// TwinCAT 3 PLC project MAIN
// ProgramVersion: 3.1.4023.0
// libraries:
//   Tc2_ModbusRTU, * (Beckhoff Automation GmbH)
//   Tc2_ModbusSrv, * (Beckhoff Automation GmbH)
//   Tc2_Standard, * (Beckhoff Automation GmbH)
//   Tc2_System, * (Beckhoff Automation GmbH)
//   Tc3_Module, * (Beckhoff Automation GmbH)
// project tree:
//   DUTs/ FUSSION.TcDUT, Inverter_SUN2000.TcDUT
//   / PlcTask.TcTTO
//   POUs/ FB_ModbusMaster_FUSSION.TcPOU, FB_ModbusMaster_Inverter.TcPOU, MAIN.TcPOU

CONFIGURATION MAIN
    RESOURCE PLC ON TwinCAT3
        TASK PlcTask(INTERVAL := T#10ms, PRIORITY := 20);
        PROGRAM MAIN WITH PlcTask : MAIN;
    END_RESOURCE
END_CONFIGURATION

// ---- DUTs/FUSSION.TcDUT
TYPE FUSSION :
STRUCT
	IPAddr		: STRING:= '127.0.0.1';
	IDSlave		: BYTE:= 255;
	TCPPort		: UINT:= 500;
	
	//--------------- LECTURA INPUT REGISTERS ---------------
	uiAddress_InputRegisters 		: ARRAY [1..19] OF UINT:= [1, 2, 3, 4, 5, 256, 257, 258, 259, 260, 261, 36864, 36865, 36866, 36867, 36868, 36869, 36870, 36871];
	uiRaw_InputRegisters 			: ARRAY [1..19] OF UINT;
	
	FSM_State_Outlet1	: UINT;
	Power_Outlet1		: UDINT;
	Energy_Outlet1		: UDINT;
	FSM_State_Outlet2	: UDINT;
	Power_Outlet2		: UDINT;
	Energy_Outlet2		: UDINT;
	Power_Phase1_Total	: UDINT;
	Power_Phase2_Total	: UDINT;
	Power_Phase3_Total	: UDINT;
	Number_Available_CPs: UDINT;
	
	//--------------- LECTURA HOLDING REGISTERS ---------------
	uiAddress_HoldingRegisters 		: ARRAY [1..18] OF WORD:= [32768,32769, 32770, 32771, 32772, 32773, 32774, 32775, 32776, 32777, 32784, 32785, 36864, 36865, 36866, 36867, 36868, 36869];
	
	uiRaw_HoldingRegisters			: ARRAY [1..18] OF UINT; // Variables leidas de Modbus para escritura en pyads
	Power_Phase1_Max_Outlet1		: UDINT;
	Power_Phase2_Max_Outlet1		: UDINT;
	Power_Phase3_Max_Outlet1		: UDINT;
	Power_Phase1_Max_Outlet2		: UDINT;
	Power_Phase2_Max_Outlet2		: UDINT;
	Power_Phase3_Max_Outlet2		: UDINT;
	Power_Phase1_Total_Max			: UDINT;
	Power_Phase2_Total_Max			: UDINT;
	Power_Phase3_Total_Max			: UDINT;
	
	uiRaw_HoldingRegisters_write	: ARRAY [1..18] OF UINT; // Variables recibidas para escritura en Modbus
		
	//Power_Phase1_Max_Outlet1_write	: UDINT;
	//Power_Phase2_Max_Outlet1_write	: UDINT;
	//Power_Phase3_Max_Outlet1_write	: UDINT;
	//Power_Phase1_Max_Outlet2_write	: UDINT;
	//Power_Phase2_Max_Outlet2_write	: UDINT;
	//Power_Phase3_Max_Outlet2_write	: UDINT;
	//Power_Phase1_Total_Max_write	: UDINT;
	//Power_Phase2_Total_Max_write	: UDINT;
	//Power_Phase3_Total_Max_write	: UDINT;
	
		
END_STRUCT
END_TYPE

// ---- DUTs/Inverter_SUN2000.TcDUT
TYPE Inverter_SUN2000 :
STRUCT
	IDSlave		: BYTE:= 255;
	TCPPort		: UINT:= 500;
	
	//--------------- LECTURA ALARMAS ---------------
	uiAddress_Alarm 		: ARRAY [1..11] OF UINT:= [50000, 50001, 50002, 50003, 50004, 50005, 50006, 50007, 50008, 50009, 50016];
	uiRaw_Alarm 			: ARRAY [1..11] OF UINT;
	
	// 50000
	Software_Ver_Unmatch_1	:	BOOL;
	Upgrade_Failed_1		:	BOOL;
	Flash_Fault_1			:	BOOL;
	// 50001
	Software_Ver_Unmatch_2	:	BOOL;
	Software_Ver_Unmatch_3	:	BOOL;
	System_Fault_1			:	BOOL;
	System_Fault_27			:	BOOL;
	Abnormal_Inv_Circuit_20	:	BOOL;
	Abnormal_Resid_Cur_1	:	BOOL;
	Cabinet_Overtemp_1		:	BOOL;
	System_Fault_28			:	BOOL;
	Fan_Fault_1				:	BOOL;
	Abnormal_SPI_Comm_1		:	BOOL;
	System_Fault_29			:	BOOL;
	//50002
	Low_Insulation_Res_1	:	BOOL;
	AFCI_Self_test_Fault_1	:	BOOL;
	DC_Arc_Fault_1			:	BOOL;
	AFCI_Self_test_Fault_2	:	BOOL;
	AFCI_Self_test_Fault_3	:	BOOL;
	System_Fault_30			:	BOOL;
	System_Fault_31			:	BOOL;
	String_3_Reversed_1		:	BOOL;
	DC_Arc_Fault_2			:	BOOL;
	DC_Arc_Fault_3			:	BOOL;
	DC_Arc_Fault_4			:	BOOL;
	System_Fault_23			:	BOOL;
	// 50003
	String_1_Reversed_1		:	BOOL;
	String_2_Reversed_1		:	BOOL;
	Abnormal_DC_Circuit_12	:	BOOL;
	String_4_Reversed_1		:	BOOL;
	String_5_Reversed_1		:	BOOL;
	String_6_Reversed_1		:	BOOL;
	High_DC_Input_Volt_1	:	BOOL;
	High_DC_Input_Volt_2	:	BOOL;
	High_DC_Input_Volt_3	:	BOOL;
	High_DC_Input_Volt_4	:	BOOL;
	Abnormal_DC_Circuit_15	:	BOOL;
	// 50004
	String_1_Reversed_2		:	BOOL;
	String_2_Reversed_2		:	BOOL;
	String_7_Reversed_1		:	BOOL;
	String_7_Reversed_2		:	BOOL;
	String_8_Reversed_1		:	BOOL;
	String_8_Reversed_2		:	BOOL;
	String_3_Reversed_2		:	BOOL;
	String_4_Reversed_2		:	BOOL;
	String_5_Reversed_2		:	BOOL;
	String_6_Reversed_2		:	BOOL;
	// 50005
	Abnormal_DC_Circuit_3	:	BOOL;
	Abnormal_Auxiliary_power_4	:	BOOL;
	Abnormal_DC_Circuit_10	:	BOOL;
	Abnormal_DC_Circuit_11	:	BOOL;
	Abnormal_DC_Circuit_30	:	BOOL;
	// 50006
	System_Fault_3			:	BOOL;
	Abnormal_Inv_Circuit_13	:	BOOL;
	Abnormal_Inv_Circuit_14	:	BOOL;
	// 50007
	Abnormal_Inv_Circuit_16	:	BOOL;
	System_Fault_21			:	BOOL;
	// 50008
	Abnormal_Grid_Volt_4	:	BOOL;
	Abnormal_Grid_Volt_16	:	BOOL;
	Frequency_Abnormal_2	:	BOOL;
	Frequency_Abnormal_4	:	BOOL;
	Abnormal_Grid_Volt_28	:	BOOL;
	Abnormal_Grid_Volt_29	:	BOOL;
	Abnormal_Ground_1		:	BOOL;
	Abnormal_Grid_Volt_26	:	BOOL;
	Frequency_Abnormal_5	:	BOOL;
	// 50009
	Abnormal_Grid_Volt_31	:	BOOL;
	Abnormal_Grid_Volt_32	:	BOOL;
	Abnormal_Grid_Volt_33	:	BOOL;
	Abnormal_Grid_Volt_19	:	BOOL;
	// 50016
	Abnormal_String_1_1		:	BOOL;
	Abnormal_String_2_1		:	BOOL;
	Abnormal_String_3_1		:	BOOL;
	Abnormal_String_4_1		:	BOOL;
	Abnormal_String_5_1		:	BOOL;
	Abnormal_String_6_1		:	BOOL;
	Abnormal_String_7_1		:	BOOL;
	Abnormal_String_8_1		:	BOOL;
	
	//--------------- LECTURA MEDIDAS ---------------
	//Falta por determinar que variables queremos medir.
	uiAddress_Signal 		: ARRAY [1..137] OF UINT:= [32001,32002,32003,32200,32262,32263,32264,32265,32266,32267,32268,32269,32270,32271,32272,32273,32274,32275,32276,32277,
														32278,32279,32280,32281,32282,32283,32284,32285,32286,32287,32288,32290,32292,32294,32296,32298,32300,32302,32304,32306,
														32314,32315,32316,32317,32320,32321,32321,32321,32322,32323,32325,32327,32343,32345,32347,32349,32351,32353,32355,32357,
														33022,33024,33026,33070,40000,40117,40118,40119,40120,40121,40122,40123,40124,40125,40133,40154,40200,40201,40232,40234,
														40235,40236,40237,42045,42047,42049,42051,42053,42055,42057,42059,42061,42063,42064,42065,42066,42067,42068,42069,42070,
														42071,42072,42074,42075,42083,42084,42085,42086,42087,42089,42090,42091,42092,42093,42094,42095,42096,42097,42101,42151,
														42152,42154,42155,42157,42158,42160,42161,42174,42300,42301,42302,42303,42304,42305,42320,42321,42333];
	uiRaw_Signal			: ARRAY [1..137] OF UINT;
END_STRUCT
END_TYPE

// ---- POUs/MAIN.TcPOU
PROGRAM MAIN
VAR
	FUSSION: FB_ModbusMaster_FUSSION;
	Inverter: FB_ModbusMaster_Inverter;
	Enable: BOOL:= TRUE;
	
	salida_pyads_InputRegisters: ARRAY[1..10] OF UINT;
	salida_pyads_HoldingsRegisters: ARRAY[1..9] OF UINT;
	entrada_pyads: ARRAY[1..9] OF UINT;
	flag_entrada_pyads: BOOL;
END_VAR

FUSSION(
	bEnable:= Enable, 
	entrada_pyads:= entrada_pyads, 
	flag_entrada_pyads:= flag_entrada_pyads, 
	salida_pyads_InputRegisters=> salida_pyads_InputRegisters, 
	salida_pyads_HoldingsRegisters=> salida_pyads_HoldingsRegisters);
	
//Inverter(bEnable:= Enable);

END_PROGRAM

// ---- POUs/FB_ModbusMaster_FUSSION.TcPOU
FUNCTION_BLOCK FB_ModbusMaster_FUSSION
VAR_INPUT
	bEnable			: BOOL;
	entrada_pyads: ARRAY[1..9] OF UINT; // Variables recibidas para escritura en Modbus
END_VAR
VAR
	iPaso			: INT;
	fbReadRegs		: FB_MBReadRegs;
	fbReadInputRegs : FB_MBReadInputRegs;
	bOcupado		: BOOL;
	
	Data_FUSSION : FUSSION;
	bAddrCount		: BYTE:= 1;
	bAddrCount2: BYTE;
	bOcupado2: BOOL;
	counter: BYTE := 1;
	fbWriteRegs: FB_MBWriteRegs;
	bOcupado3: BOOL;
	
END_VAR
VAR_OUTPUT
	salida_pyads_InputRegisters: ARRAY[1..10] OF UINT;
	salida_pyads_HoldingsRegisters: ARRAY[1..9] OF UINT;
END_VAR
VAR_IN_OUT
	flag_entrada_pyads: BOOL;
END_VAR

CASE iPaso OF
0:	//Inicio
	fbReadRegs(bExecute := FALSE);
	fbReadInputRegs(bExecute := FALSE);
	IF bEnable THEN
		iPaso := 1;
	END_IF

1: //Lectura Input Registers
	fbReadInputRegs(
			sIPAddr		:= Data_FUSSION.IPAddr, 
			nTCPPort	:= Data_FUSSION.TCPPort, 
			nUnitID		:= Data_FUSSION.IDSlave, 
			nQuantity	:= 1, 
			nMBAddr		:= Data_FUSSION.uiAddress_InputRegisters[bAddrCount],
			cbLength	:= SIZEOF(Data_FUSSION.uiRaw_InputRegisters[bAddrCount]),
			pDestAddr	:= ADR(Data_FUSSION.uiRaw_InputRegisters[bAddrCount]), 
			bExecute	:= TRUE, 
			tTimeout	:= T#1S, 
			bBusy		=> bOcupado, 
			bError		=> , 
			nErrId		=> , 
			cbRead		=> );
	IF NOT bOcupado THEN
		fbReadInputRegs(bExecute := FALSE);
		bAddrCount := bAddrCount+1;
		IF bAddrCount > 19 THEN
			bAddrCount := 1;
			bAddrCount2 := 1;
			iPaso := 4;	
		END_IF
	END_IF
	
3: //Lectura Holding Registers
	fbReadRegs(
		sIPAddr		:= Data_FUSSION.IPAddr, 
		nTCPPort	:= Data_FUSSION.TCPPort, 
		nUnitID		:= Data_FUSSION.IDSlave, 
		nQuantity	:= 1,
		nMBAddr		:= Data_FUSSION.uiAddress_HoldingRegisters[bAddrCount2],
		cbLength	:= SIZEOF(Data_FUSSION.uiRaw_HoldingRegisters[bAddrCount2]), 
		pDestAddr	:= ADR(Data_FUSSION.uiRaw_HoldingRegisters[bAddrCount2]), 
		bExecute	:= TRUE, 
		tTimeout	:= T#1S, 
		bBusy		=> bOcupado2, 
		bError		=> , 
		nErrId		=> , 
		cbRead		=> );
	IF NOT bOcupado2 THEN
		fbReadRegs(bExecute := FALSE);
		bAddrCount2 := bAddrCount2+1;
			IF bAddrCount2 > 18 THEN
				bAddrCount2 := 1;
				iPaso := 4;	
			END_IF
	END_IF

4: //Escalado Input Registers
	Data_FUSSION.FSM_State_Outlet1 		:= Data_FUSSION.uiRaw_InputRegisters[1]; // Little
	Data_FUSSION.Power_Outlet1			:= SHL(Data_FUSSION.uiRaw_InputRegisters[3], 8) + Data_FUSSION.uiRaw_InputRegisters[2];
	Data_FUSSION.Energy_Outlet1			:= SHL(Data_FUSSION.uiRaw_InputRegisters[5], 8) + Data_FUSSION.uiRaw_InputRegisters[4];
	Data_FUSSION.FSM_State_Outlet2		:= SHL(Data_FUSSION.uiRaw_InputRegisters[7], 8) + Data_FUSSION.uiRaw_InputRegisters[6];
	Data_FUSSION.Power_Outlet2			:= SHL(Data_FUSSION.uiRaw_InputRegisters[9], 8) + Data_FUSSION.uiRaw_InputRegisters[8];
	Data_FUSSION.Energy_Outlet2			:= SHL(Data_FUSSION.uiRaw_InputRegisters[11], 8) + Data_FUSSION.uiRaw_InputRegisters[10];
	Data_FUSSION.Power_Phase1_Total		:= SHL(Data_FUSSION.uiRaw_InputRegisters[12], 8) + Data_FUSSION.uiRaw_InputRegisters[13]; // Big
	Data_FUSSION.Power_Phase2_Total		:= SHL(Data_FUSSION.uiRaw_InputRegisters[14], 8) + Data_FUSSION.uiRaw_InputRegisters[15];
	Data_FUSSION.Power_Phase3_Total		:= SHL(Data_FUSSION.uiRaw_InputRegisters[16], 8) + Data_FUSSION.uiRaw_InputRegisters[17];
	Data_FUSSION.Number_Available_CPs 	:= SHL(Data_FUSSION.uiRaw_InputRegisters[18], 8) + Data_FUSSION.uiRaw_InputRegisters[19];
	
	//Temporales pyads
	salida_pyads_InputRegisters[1] 		:= Data_FUSSION.uiRaw_InputRegisters[1]; // Little
	salida_pyads_InputRegisters[2]		:= SHL(Data_FUSSION.uiRaw_InputRegisters[3], 8) + Data_FUSSION.uiRaw_InputRegisters[2];
	salida_pyads_InputRegisters[3]		:= SHL(Data_FUSSION.uiRaw_InputRegisters[5], 8) + Data_FUSSION.uiRaw_InputRegisters[4];
	salida_pyads_InputRegisters[4]		:= SHL(Data_FUSSION.uiRaw_InputRegisters[7], 8) + Data_FUSSION.uiRaw_InputRegisters[6];
	salida_pyads_InputRegisters[5]		:= SHL(Data_FUSSION.uiRaw_InputRegisters[9], 8) + Data_FUSSION.uiRaw_InputRegisters[8];
	salida_pyads_InputRegisters[6]		:= SHL(Data_FUSSION.uiRaw_InputRegisters[11], 8) + Data_FUSSION.uiRaw_InputRegisters[10];
	salida_pyads_InputRegisters[7]		:= SHL(Data_FUSSION.uiRaw_InputRegisters[12], 8) + Data_FUSSION.uiRaw_InputRegisters[13]; // Big
	salida_pyads_InputRegisters[8]		:= SHL(Data_FUSSION.uiRaw_InputRegisters[14], 8) + Data_FUSSION.uiRaw_InputRegisters[15];
	salida_pyads_InputRegisters[9]		:= SHL(Data_FUSSION.uiRaw_InputRegisters[16], 8) + Data_FUSSION.uiRaw_InputRegisters[17];
	salida_pyads_InputRegisters[10]	 	:= SHL(Data_FUSSION.uiRaw_InputRegisters[18], 8) + Data_FUSSION.uiRaw_InputRegisters[19];

	iPaso := 6;
	
5: //Escalado Holding Registers
	Data_FUSSION.Power_Phase1_Max_Outlet1	:= SHL(Data_FUSSION.uiRaw_HoldingRegisters[2], 8) + Data_FUSSION.uiRaw_HoldingRegisters[1]; // Little
	Data_FUSSION.Power_Phase2_Max_Outlet1	:= SHL(Data_FUSSION.uiRaw_HoldingRegisters[4], 8) + Data_FUSSION.uiRaw_HoldingRegisters[3];
	Data_FUSSION.Power_Phase3_Max_Outlet1	:= SHL(Data_FUSSION.uiRaw_HoldingRegisters[6], 8) + Data_FUSSION.uiRaw_HoldingRegisters[5];
	Data_FUSSION.Power_Phase1_Max_Outlet2	:= SHL(Data_FUSSION.uiRaw_HoldingRegisters[8], 8) + Data_FUSSION.uiRaw_HoldingRegisters[7];
	Data_FUSSION.Power_Phase2_Max_Outlet2	:= SHL(Data_FUSSION.uiRaw_HoldingRegisters[10], 8) + Data_FUSSION.uiRaw_HoldingRegisters[9];
	Data_FUSSION.Power_Phase3_Max_Outlet2	:= SHL(Data_FUSSION.uiRaw_HoldingRegisters[12], 8) + Data_FUSSION.uiRaw_HoldingRegisters[11];
	Data_FUSSION.Power_Phase1_Total_Max		:= SHL(Data_FUSSION.uiRaw_HoldingRegisters[13], 8) + Data_FUSSION.uiRaw_HoldingRegisters[14]; // Big
	Data_FUSSION.Power_Phase2_Total_Max		:= SHL(Data_FUSSION.uiRaw_HoldingRegisters[15], 8) + Data_FUSSION.uiRaw_HoldingRegisters[16];
	Data_FUSSION.Power_Phase3_Total_Max		:= SHL(Data_FUSSION.uiRaw_HoldingRegisters[17], 8) + Data_FUSSION.uiRaw_HoldingRegisters[18];
	
	//Temporales pyads
	salida_pyads_HoldingsRegisters[1]		:= SHL(Data_FUSSION.uiRaw_HoldingRegisters[2], 8) + Data_FUSSION.uiRaw_HoldingRegisters[1]; // Little
	salida_pyads_HoldingsRegisters[2]		:= SHL(Data_FUSSION.uiRaw_HoldingRegisters[4], 8) + Data_FUSSION.uiRaw_HoldingRegisters[3];
	salida_pyads_HoldingsRegisters[3]		:= SHL(Data_FUSSION.uiRaw_HoldingRegisters[6], 8) + Data_FUSSION.uiRaw_HoldingRegisters[5];
	salida_pyads_HoldingsRegisters[4]		:= SHL(Data_FUSSION.uiRaw_HoldingRegisters[8], 8) + Data_FUSSION.uiRaw_HoldingRegisters[7];
	salida_pyads_HoldingsRegisters[5]		:= SHL(Data_FUSSION.uiRaw_HoldingRegisters[10], 8) + Data_FUSSION.uiRaw_HoldingRegisters[9];
	salida_pyads_HoldingsRegisters[6]		:= SHL(Data_FUSSION.uiRaw_HoldingRegisters[12], 8) + Data_FUSSION.uiRaw_HoldingRegisters[11];
	salida_pyads_HoldingsRegisters[7]		:= SHL(Data_FUSSION.uiRaw_HoldingRegisters[13], 8) + Data_FUSSION.uiRaw_HoldingRegisters[14]; // Big
	salida_pyads_HoldingsRegisters[8]		:= SHL(Data_FUSSION.uiRaw_HoldingRegisters[15], 8) + Data_FUSSION.uiRaw_HoldingRegisters[16];
	salida_pyads_HoldingsRegisters[9]		:= SHL(Data_FUSSION.uiRaw_HoldingRegisters[17], 8) + Data_FUSSION.uiRaw_HoldingRegisters[18];

	iPaso := 6;
	
6: //Envío pyads

	iPaso := 7;
	
7: //Recepción pyads

	iPaso := 8;
	
8: //Escalado Holding Registers para escritura
	IF flag_entrada_pyads = 1 THEN
		Data_FUSSION.uiRaw_HoldingRegisters_write[1]	:= UDINT_TO_UINT(entrada_pyads[1]); // Little
		Data_FUSSION.uiRaw_HoldingRegisters_write[2]	:= UDINT_TO_UINT(SHR(entrada_pyads[1], 8));
		Data_FUSSION.uiRaw_HoldingRegisters_write[3]	:= UDINT_TO_UINT(entrada_pyads[2]);
		Data_FUSSION.uiRaw_HoldingRegisters_write[4]	:= UDINT_TO_UINT(SHR(entrada_pyads[2], 8));
		Data_FUSSION.uiRaw_HoldingRegisters_write[5]	:= UDINT_TO_UINT(entrada_pyads[3]);
		Data_FUSSION.uiRaw_HoldingRegisters_write[6]	:= UDINT_TO_UINT(SHR(entrada_pyads[3], 8));
		Data_FUSSION.uiRaw_HoldingRegisters_write[7]	:= UDINT_TO_UINT(entrada_pyads[4]);
		Data_FUSSION.uiRaw_HoldingRegisters_write[8]	:= UDINT_TO_UINT(SHR(entrada_pyads[4], 8));
		Data_FUSSION.uiRaw_HoldingRegisters_write[9]	:= UDINT_TO_UINT(entrada_pyads[5]);
		Data_FUSSION.uiRaw_HoldingRegisters_write[10]	:= UDINT_TO_UINT(SHR(entrada_pyads[5], 8));
		Data_FUSSION.uiRaw_HoldingRegisters_write[11]	:= UDINT_TO_UINT(entrada_pyads[6]);
		Data_FUSSION.uiRaw_HoldingRegisters_write[12]	:= UDINT_TO_UINT(SHR(entrada_pyads[6], 8));
		Data_FUSSION.uiRaw_HoldingRegisters_write[13]	:= UDINT_TO_UINT(SHR(entrada_pyads[7], 8)); // Big
		Data_FUSSION.uiRaw_HoldingRegisters_write[14]	:= UDINT_TO_UINT(entrada_pyads[7]);
		Data_FUSSION.uiRaw_HoldingRegisters_write[15]	:= UDINT_TO_UINT(SHR(entrada_pyads[8], 8));
		Data_FUSSION.uiRaw_HoldingRegisters_write[16]	:= UDINT_TO_UINT(entrada_pyads[8]);
		Data_FUSSION.uiRaw_HoldingRegisters_write[17]	:= UDINT_TO_UINT(SHR(entrada_pyads[9], 8));
		Data_FUSSION.uiRaw_HoldingRegisters_write[18]	:= UDINT_TO_UINT(entrada_pyads[9]);	
	
		IF counter <= 18 THEN
			//IF NOT (Data_FUSSION.uiRaw_HoldingRegisters_write[counter] = Data_FUSSION.uiRaw_HoldingRegisters[counter]) THEN
				fbWriteRegs(
					sIPAddr		:= Data_FUSSION.IPAddr, 
					nTCPPort	:= Data_FUSSION.TCPPort, 
					nUnitID		:= Data_FUSSION.IDSlave, 
					nQuantity	:= 1,
					nMBAddr		:= Data_FUSSION.uiAddress_HoldingRegisters[counter],
					cbLength	:= SIZEOF(Data_FUSSION.uiRaw_HoldingRegisters_write[counter]),  
					pSrcAddr	:= ADR(Data_FUSSION.uiRaw_HoldingRegisters_write[counter]), 
					bExecute	:= TRUE, 
					tTimeout	:= T#1S, 
					bBusy		=> bOcupado3, 
					bError		=> , 
					nErrId		=> );
				IF NOT bOcupado3 THEN
					fbWriteRegs(bExecute := FALSE);
					counter := counter+1;
					IF counter >= 18 THEN
						counter := 1;
						flag_entrada_pyads:= 0;
						iPaso := 0;	
					END_IF
				END_IF
			//END_IF
		END_IF	
	
	ELSE
		iPaso:= 0;
	END_IF
END_CASE

END_FUNCTION_BLOCK

// ---- POUs/FB_ModbusMaster_Inverter.TcPOU
FUNCTION_BLOCK FB_ModbusMaster_Inverter
VAR_INPUT
	bEnable			: BOOL;
END_VAR
VAR_OUTPUT
END_VAR
VAR
	fbModbusRtuMasterV2: ModbusRtuMasterV2_KL6x22B;
	bAddrCount		: BYTE:= 1;
	
	Data_Inverter_SUN2000	: Inverter_SUN2000;
	iPaso: INT;
END_VAR

CASE iPaso OF
0:	//Inicio
	IF bEnable THEN
		iPaso := 1;
	END_IF

1: //Lectura de alarmas
	fbModbusRtuMasterV2.ReadInputRegs(
		UnitID:= Data_Inverter_SUN2000.IDSlave,
		Quantity:= 1,
		MBAddr:= Data_Inverter_SUN2000.uiAddress_Alarm[bAddrCount],
		cbLength:= SIZEOF(Data_Inverter_SUN2000.uiRaw_Alarm[bAddrCount]),
		pMemoryAddr:= ADR(Data_Inverter_SUN2000.uiRaw_Alarm[bAddrCount]), 
		Timeout:= T#1S,
		//AuxQuantity:= , //solo para funcion modbus 23
		//AuxMBAddr:= , 	//solo para funcion modbus 23
		//AuxcbLength:= , //solo para funcion modbus 23
		//pAuxMemoryAddr:= , //solo para funcion modbus 23
		Execute:= TRUE);
		
	IF NOT fbModbusRtuMasterV2.BUSY THEN
		bAddrCount := bAddrCount+1;
		IF bAddrCount > 11 THEN
			bAddrCount := 1;
			iPaso := 3;	
		END_IF
	END_IF
	
3: //Lectura de medidas
	fbModbusRtuMasterV2.ReadInputRegs(
		UnitID:= Data_Inverter_SUN2000.IDSlave,
		Quantity:= 1,
		MBAddr:= Data_Inverter_SUN2000.uiAddress_Signal[bAddrCount],
		cbLength:= SIZEOF(Data_Inverter_SUN2000.uiRaw_Signal[bAddrCount]),
		pMemoryAddr:= ADR(Data_Inverter_SUN2000.uiRaw_Signal[bAddrCount]), 
		Timeout:= T#1S,
		//AuxQuantity:= , //solo para funcion modbus 23
		//AuxMBAddr:= , 	//solo para funcion modbus 23
		//AuxcbLength:= , //solo para funcion modbus 23
		//pAuxMemoryAddr:= , //solo para funcion modbus 23
		Execute:= TRUE);
		
	IF NOT fbModbusRtuMasterV2.BUSY THEN
		bAddrCount := bAddrCount+1;
		IF bAddrCount > 11 THEN
			bAddrCount := 1;
			iPaso := 4;	
		END_IF
	END_IF
	
4: //Escalado de variables de alarma
	Data_Inverter_SUN2000.Software_Ver_Unmatch_1	:= UINT_TO_BOOL(Data_Inverter_SUN2000.uiRaw_Alarm[1] AND 16#0A);
	Data_Inverter_SUN2000.Upgrade_Failed_1			:= UINT_TO_BOOL(Data_Inverter_SUN2000.uiRaw_Alarm[1] AND 16#0B);
	Data_Inverter_SUN2000.Flash_Fault_1				:= UINT_TO_BOOL(Data_Inverter_SUN2000.uiRaw_Alarm[1] AND 16#0C);
	
	Data_Inverter_SUN2000.Software_Ver_Unmatch_2	:= UINT_TO_BOOL(Data_Inverter_SUN2000.uiRaw_Alarm[2] AND 16#01);
	Data_Inverter_SUN2000.Software_Ver_Unmatch_3	:= UINT_TO_BOOL(Data_Inverter_SUN2000.uiRaw_Alarm[2] AND 16#02);
	Data_Inverter_SUN2000.System_Fault_1			:= UINT_TO_BOOL(Data_Inverter_SUN2000.uiRaw_Alarm[2] AND 16#03);
	Data_Inverter_SUN2000.System_Fault_27			:= UINT_TO_BOOL(Data_Inverter_SUN2000.uiRaw_Alarm[2] AND 16#04);
	Data_Inverter_SUN2000.Abnormal_Inv_Circuit_20	:= UINT_TO_BOOL(Data_Inverter_SUN2000.uiRaw_Alarm[2] AND 16#06);
	Data_Inverter_SUN2000.Abnormal_Resid_Cur_1		:= UINT_TO_BOOL(Data_Inverter_SUN2000.uiRaw_Alarm[2] AND 16#07);
	Data_Inverter_SUN2000.Cabinet_Overtemp_1		:= UINT_TO_BOOL(Data_Inverter_SUN2000.uiRaw_Alarm[2] AND 16#08);
	Data_Inverter_SUN2000.System_Fault_28			:= UINT_TO_BOOL(Data_Inverter_SUN2000.uiRaw_Alarm[2] AND 16#0A);
	Data_Inverter_SUN2000.Fan_Fault_1				:= UINT_TO_BOOL(Data_Inverter_SUN2000.uiRaw_Alarm[2] AND 16#0B);
	Data_Inverter_SUN2000.Abnormal_SPI_Comm_1		:= UINT_TO_BOOL(Data_Inverter_SUN2000.uiRaw_Alarm[2] AND 16#0C);
	Data_Inverter_SUN2000.System_Fault_29			:= UINT_TO_BOOL(Data_Inverter_SUN2000.uiRaw_Alarm[2] AND 16#0E);
	
	Data_Inverter_SUN2000.Low_Insulation_Res_1		:= UINT_TO_BOOL(Data_Inverter_SUN2000.uiRaw_Alarm[3] AND 16#00);
	Data_Inverter_SUN2000.AFCI_Self_test_Fault_1	:= UINT_TO_BOOL(Data_Inverter_SUN2000.uiRaw_Alarm[3] AND 16#01);
	Data_Inverter_SUN2000.DC_Arc_Fault_1			:= UINT_TO_BOOL(Data_Inverter_SUN2000.uiRaw_Alarm[3] AND 16#02);
	Data_Inverter_SUN2000.AFCI_Self_test_Fault_2	:= UINT_TO_BOOL(Data_Inverter_SUN2000.uiRaw_Alarm[3] AND 16#03);
	Data_Inverter_SUN2000.AFCI_Self_test_Fault_3	:= UINT_TO_BOOL(Data_Inverter_SUN2000.uiRaw_Alarm[3] AND 16#04);
	Data_Inverter_SUN2000.System_Fault_30			:= UINT_TO_BOOL(Data_Inverter_SUN2000.uiRaw_Alarm[3] AND 16#07);
	Data_Inverter_SUN2000.System_Fault_31			:= UINT_TO_BOOL(Data_Inverter_SUN2000.uiRaw_Alarm[3] AND 16#08);
	Data_Inverter_SUN2000.String_3_Reversed_1		:= UINT_TO_BOOL(Data_Inverter_SUN2000.uiRaw_Alarm[3] AND 16#09);
	Data_Inverter_SUN2000.DC_Arc_Fault_2			:= UINT_TO_BOOL(Data_Inverter_SUN2000.uiRaw_Alarm[3] AND 16#0C);
	Data_Inverter_SUN2000.DC_Arc_Fault_3			:= UINT_TO_BOOL(Data_Inverter_SUN2000.uiRaw_Alarm[3] AND 16#0D);
	Data_Inverter_SUN2000.DC_Arc_Fault_4			:= UINT_TO_BOOL(Data_Inverter_SUN2000.uiRaw_Alarm[3] AND 16#0E);
	Data_Inverter_SUN2000.System_Fault_23			:= UINT_TO_BOOL(Data_Inverter_SUN2000.uiRaw_Alarm[3] AND 16#0F);
	
	Data_Inverter_SUN2000.String_1_Reversed_1		:= UINT_TO_BOOL(Data_Inverter_SUN2000.uiRaw_Alarm[4] AND 16#01);
	Data_Inverter_SUN2000.String_2_Reversed_1		:= UINT_TO_BOOL(Data_Inverter_SUN2000.uiRaw_Alarm[4] AND 16#02);
	Data_Inverter_SUN2000.Abnormal_DC_Circuit_12	:= UINT_TO_BOOL(Data_Inverter_SUN2000.uiRaw_Alarm[4] AND 16#03);
	Data_Inverter_SUN2000.String_4_Reversed_1		:= UINT_TO_BOOL(Data_Inverter_SUN2000.uiRaw_Alarm[4] AND 16#06);
	Data_Inverter_SUN2000.String_5_Reversed_1		:= UINT_TO_BOOL(Data_Inverter_SUN2000.uiRaw_Alarm[4] AND 16#07);
	Data_Inverter_SUN2000.String_6_Reversed_1		:= UINT_TO_BOOL(Data_Inverter_SUN2000.uiRaw_Alarm[4] AND 16#08);
	Data_Inverter_SUN2000.High_DC_Input_Volt_1		:= UINT_TO_BOOL(Data_Inverter_SUN2000.uiRaw_Alarm[4] AND 16#09);
	Data_Inverter_SUN2000.High_DC_Input_Volt_2		:= UINT_TO_BOOL(Data_Inverter_SUN2000.uiRaw_Alarm[4] AND 16#0A);
	Data_Inverter_SUN2000.High_DC_Input_Volt_3		:= UINT_TO_BOOL(Data_Inverter_SUN2000.uiRaw_Alarm[4] AND 16#0B);
	Data_Inverter_SUN2000.High_DC_Input_Volt_4		:= UINT_TO_BOOL(Data_Inverter_SUN2000.uiRaw_Alarm[4] AND 16#0C);
	Data_Inverter_SUN2000.Abnormal_DC_Circuit_15	:= UINT_TO_BOOL(Data_Inverter_SUN2000.uiRaw_Alarm[4] AND 16#0F);
	
	Data_Inverter_SUN2000.String_1_Reversed_2		:= UINT_TO_BOOL(Data_Inverter_SUN2000.uiRaw_Alarm[5] AND 16#02);
	Data_Inverter_SUN2000.String_2_Reversed_2		:= UINT_TO_BOOL(Data_Inverter_SUN2000.uiRaw_Alarm[5] AND 16#03);
	Data_Inverter_SUN2000.String_7_Reversed_1		:= UINT_TO_BOOL(Data_Inverter_SUN2000.uiRaw_Alarm[5] AND 16#04);
	Data_Inverter_SUN2000.String_7_Reversed_2		:= UINT_TO_BOOL(Data_Inverter_SUN2000.uiRaw_Alarm[5] AND 16#05);
	Data_Inverter_SUN2000.String_8_Reversed_1		:= UINT_TO_BOOL(Data_Inverter_SUN2000.uiRaw_Alarm[5] AND 16#06);
	Data_Inverter_SUN2000.String_8_Reversed_2		:= UINT_TO_BOOL(Data_Inverter_SUN2000.uiRaw_Alarm[5] AND 16#07);
	Data_Inverter_SUN2000.String_3_Reversed_2		:= UINT_TO_BOOL(Data_Inverter_SUN2000.uiRaw_Alarm[5] AND 16#0C);
	Data_Inverter_SUN2000.String_4_Reversed_2		:= UINT_TO_BOOL(Data_Inverter_SUN2000.uiRaw_Alarm[5] AND 16#0D);
	Data_Inverter_SUN2000.String_5_Reversed_2		:= UINT_TO_BOOL(Data_Inverter_SUN2000.uiRaw_Alarm[5] AND 16#0E);
	Data_Inverter_SUN2000.String_6_Reversed_2		:= UINT_TO_BOOL(Data_Inverter_SUN2000.uiRaw_Alarm[5] AND 16#0F);
	
	Data_Inverter_SUN2000.Abnormal_DC_Circuit_3		:= UINT_TO_BOOL(Data_Inverter_SUN2000.uiRaw_Alarm[6] AND 16#01);
	Data_Inverter_SUN2000.Abnormal_Auxiliary_power_4	:= UINT_TO_BOOL(Data_Inverter_SUN2000.uiRaw_Alarm[6] AND 16#02);
	Data_Inverter_SUN2000.Abnormal_DC_Circuit_10	:= UINT_TO_BOOL(Data_Inverter_SUN2000.uiRaw_Alarm[6] AND 16#04);
	Data_Inverter_SUN2000.Abnormal_DC_Circuit_11	:= UINT_TO_BOOL(Data_Inverter_SUN2000.uiRaw_Alarm[6] AND 16#05);
	Data_Inverter_SUN2000.Abnormal_DC_Circuit_30	:= UINT_TO_BOOL(Data_Inverter_SUN2000.uiRaw_Alarm[6] AND 16#06);
	
	Data_Inverter_SUN2000.System_Fault_3			:= UINT_TO_BOOL(Data_Inverter_SUN2000.uiRaw_Alarm[7] AND 16#06);
	Data_Inverter_SUN2000.Abnormal_Inv_Circuit_13	:= UINT_TO_BOOL(Data_Inverter_SUN2000.uiRaw_Alarm[7] AND 16#0A);
	Data_Inverter_SUN2000.Abnormal_Inv_Circuit_14	:= UINT_TO_BOOL(Data_Inverter_SUN2000.uiRaw_Alarm[7] AND 16#0C);
	
	Data_Inverter_SUN2000.Abnormal_Inv_Circuit_16	:= UINT_TO_BOOL(Data_Inverter_SUN2000.uiRaw_Alarm[8] AND 16#01);
	Data_Inverter_SUN2000.System_Fault_21			:= UINT_TO_BOOL(Data_Inverter_SUN2000.uiRaw_Alarm[8] AND 16#05);
	
	Data_Inverter_SUN2000.Abnormal_Grid_Volt_4		:= UINT_TO_BOOL(Data_Inverter_SUN2000.uiRaw_Alarm[9] AND 16#00);
	Data_Inverter_SUN2000.Abnormal_Grid_Volt_16		:= UINT_TO_BOOL(Data_Inverter_SUN2000.uiRaw_Alarm[9] AND 16#03);
	Data_Inverter_SUN2000.Frequency_Abnormal_2		:= UINT_TO_BOOL(Data_Inverter_SUN2000.uiRaw_Alarm[9] AND 16#06);
	Data_Inverter_SUN2000.Frequency_Abnormal_4		:= UINT_TO_BOOL(Data_Inverter_SUN2000.uiRaw_Alarm[9] AND 16#07);
	Data_Inverter_SUN2000.Abnormal_Grid_Volt_28		:= UINT_TO_BOOL(Data_Inverter_SUN2000.uiRaw_Alarm[9] AND 16#08);
	Data_Inverter_SUN2000.Abnormal_Grid_Volt_29		:= UINT_TO_BOOL(Data_Inverter_SUN2000.uiRaw_Alarm[9] AND 16#09);
	Data_Inverter_SUN2000.Abnormal_Ground_1			:= UINT_TO_BOOL(Data_Inverter_SUN2000.uiRaw_Alarm[9] AND 16#0A);
	Data_Inverter_SUN2000.Abnormal_Grid_Volt_26		:= UINT_TO_BOOL(Data_Inverter_SUN2000.uiRaw_Alarm[9] AND 16#0B);
	Data_Inverter_SUN2000.Frequency_Abnormal_5		:= UINT_TO_BOOL(Data_Inverter_SUN2000.uiRaw_Alarm[9] AND 16#0C);
	
	Data_Inverter_SUN2000.Abnormal_Grid_Volt_31		:= UINT_TO_BOOL(Data_Inverter_SUN2000.uiRaw_Alarm[10] AND 16#00);
	Data_Inverter_SUN2000.Abnormal_Grid_Volt_32		:= UINT_TO_BOOL(Data_Inverter_SUN2000.uiRaw_Alarm[10] AND 16#01);
	Data_Inverter_SUN2000.Abnormal_Grid_Volt_33		:= UINT_TO_BOOL(Data_Inverter_SUN2000.uiRaw_Alarm[10] AND 16#02);
	Data_Inverter_SUN2000.Abnormal_Grid_Volt_19		:= UINT_TO_BOOL(Data_Inverter_SUN2000.uiRaw_Alarm[10] AND 16#08);
	
	Data_Inverter_SUN2000.Abnormal_String_1_1		:= UINT_TO_BOOL(Data_Inverter_SUN2000.uiRaw_Alarm[11] AND 16#00);
	Data_Inverter_SUN2000.Abnormal_String_2_1		:= UINT_TO_BOOL(Data_Inverter_SUN2000.uiRaw_Alarm[11] AND 16#01);
	Data_Inverter_SUN2000.Abnormal_String_3_1		:= UINT_TO_BOOL(Data_Inverter_SUN2000.uiRaw_Alarm[11] AND 16#02);
	Data_Inverter_SUN2000.Abnormal_String_4_1		:= UINT_TO_BOOL(Data_Inverter_SUN2000.uiRaw_Alarm[11] AND 16#03);
	Data_Inverter_SUN2000.Abnormal_String_5_1		:= UINT_TO_BOOL(Data_Inverter_SUN2000.uiRaw_Alarm[11] AND 16#04);
	Data_Inverter_SUN2000.Abnormal_String_6_1		:= UINT_TO_BOOL(Data_Inverter_SUN2000.uiRaw_Alarm[11] AND 16#05);
	Data_Inverter_SUN2000.Abnormal_String_7_1		:= UINT_TO_BOOL(Data_Inverter_SUN2000.uiRaw_Alarm[11] AND 16#06);
	Data_Inverter_SUN2000.Abnormal_String_8_1		:= UINT_TO_BOOL(Data_Inverter_SUN2000.uiRaw_Alarm[11] AND 16#07);	

	iPaso := 5;
	
5: //Escalado de variables de medida

	iPaso := 0;
	
END_CASE

END_FUNCTION_BLOCK
